{attribute addProperty BoxType "EPP1816-0003-0016"}
{attribute addProperty Id "DIG_Inputs_ChannelAT %I*ARRAY[0..1] OF DIG_Inputs_Channel_C8B92B82160200WcStateAT %I*WcState_98A4DF7520.250InfoDataAT %I*InfoData_BC63D37F80100"}
{attribute addProperty CRC "2428839517"}
{attribute addProperty SizeInBites "242"}
{attribute addProperty SizeInBytes "30.25"}
TYPE EPP1816_8758F163 :
STRUCT
	{attribute addProperty Name "DIG_Inputs_Channel"}
	DIG_Inputs_Channel : ARRAY[0..1] OF DIG_Inputs_Channel_C8B92B82;
	{attribute addProperty Name "WcState"}
	WcState : WcState_98A4DF75;
	{attribute addProperty Name "InfoData"}
	InfoData : InfoData_BC63D37F;
END_STRUCT
END_TYPE

(* stored: Version 1.2.0.0, ProductVersion 3.1.4024.9
   DUT EPP1816_8758F163: Id {9fd56ad4-2ac0-46c4-9201-1756d3e7f736} *)
